INTERFACE INTERNAL I_Sinamics

METHOD GetAcylicParameter : BOOL
VAR_INPUT
	stParameter : POINTER TO ST_PROFIdriveParam;
END_VAR
END_METHOD

METHOD SetAcylicParameter : BOOL
VAR_INPUT
	pParameter :  POINTER TO ST_PROFIdriveParam;
END_VAR
END_METHOD

METHOD TrigSafetyStop
END_METHOD

END_INTERFACE

(* stored: Version 1.1.0.1, ProductVersion 3.1.4024.12
   Itf I_Sinamics: Id {d54f4273-798f-0e19-24f9-643cada08425}
   Method GetAcylicParameter: Id {86dd38db-7016-0f65-1371-9bbb76d19c52}
   Method SetAcylicParameter: Id {d0b9d42b-f220-0d14-2101-0bf8636436c3}
   Method TrigSafetyStop: Id {5fc77642-6361-07b9-0f66-de56ef1c951a} *)
